TYPE ST_BoolHmi :
STRUCT
	Enabled: BOOL;
	PlcToHmi: BOOL;
	HmiToPlc: BOOL;
END_STRUCT
END_TYPE

(* stored: Version 1.1.0.1, ProductVersion 3.1.4024.11
   DUT ST_BoolHmi: Id {532a3cf3-4e50-47bd-8a52-1905ab6cc62f} *)
